(* IEC 61131-3 sources: ml2plc/benchmarks/st (part 26) *)

VAR
    (* Merged variables from all regions *)
    buffer_0 : ARRAY[0..63] OF REAL;
    buffer_1 : ARRAY[0..63] OF REAL;
    buffer_2 : ARRAY[0..63] OF REAL;

    (* Temporary computation variables *)
    i : DINT;
    j : DINT;
    t : DINT;
    sum : REAL;
    (* Computation helpers *)
    max_val : REAL;
    exp_val : REAL;
    exp_sum : REAL;
    (* Spatial loop variables *)
    oc : DINT;
    oh : DINT;
    ow : DINT;
    ic : DINT;
    kh : DINT;
    kw : DINT;
    ih : DINT;
    iw : DINT;
END_VAR

(* Forward pass execution *)

(* Region: r0 [ACYCLIC] *)
(* Acyclic Region r0 *)
(* Layer 0: Fused Linear + RELU *)
FOR j := 0 TO 63 DO
    sum := 0.0;
    FOR i := 0 TO 0 DO
        sum := sum + input_data * weights_0[i * 64 + j];
    END_FOR;
buffer_0[j] := MAX(sum + bias_0[j], 0.0);
END_FOR;

(* Layer 1: Fused Linear + RELU *)
FOR j := 0 TO 63 DO
    sum := 0.0;
    FOR i := 0 TO 63 DO
        sum := sum + buffer_0[i] * weights_1[i * 64 + j];
    END_FOR;
buffer_2[j] := MAX(sum + bias_1[j], 0.0);
END_FOR;

(* Layer 2: MatMul *)
FOR j := 0 TO 63 DO
    sum := 0.0;
    FOR i := 0 TO 63 DO
        sum := sum + buffer_2[i] * weights_2[i * 64 + j];
    END_FOR;
buffer_1[j] := sum;
END_FOR;

(* Layer 3: Add (Bias) *)
FOR i := 0 TO 63 DO
    buffer_2[i] := buffer_1[i] + bias_3[i];
END_FOR;

(* Layer 4: Add (Element-wise) *)
FOR i := 0 TO 63 DO
    buffer_1[i] := buffer_2[i] + buffer_0[i];
END_FOR;

(* Layer 5: Activation (RELU) *)
FOR i := 0 TO 63 DO
    buffer_0[i] := MAX(buffer_1[i], 0.0);
END_FOR;

(* Layer 6: Fused Linear + RELU *)
FOR j := 0 TO 63 DO
    sum := 0.0;
    FOR i := 0 TO 63 DO
        sum := sum + buffer_0[i] * weights_6[i * 64 + j];
    END_FOR;
buffer_2[j] := MAX(sum + bias_6[j], 0.0);
END_FOR;

(* Layer 7: MatMul *)
FOR j := 0 TO 63 DO
    sum := 0.0;
    FOR i := 0 TO 63 DO
        sum := sum + buffer_2[i] * weights_7[i * 64 + j];
    END_FOR;
buffer_1[j] := sum;
END_FOR;

(* Layer 8: Add (Bias) *)
FOR i := 0 TO 63 DO
    buffer_2[i] := buffer_1[i] + bias_8[i];
END_FOR;

(* Layer 9: Add (Element-wise) *)
FOR i := 0 TO 63 DO
    buffer_1[i] := buffer_2[i] + buffer_0[i];
END_FOR;

(* Layer 10: Activation (RELU) *)
FOR i := 0 TO 63 DO
    buffer_0[i] := MAX(buffer_1[i], 0.0);
END_FOR;

(* Layer 11: Fused Linear + RELU *)
FOR j := 0 TO 63 DO
    sum := 0.0;
    FOR i := 0 TO 63 DO
        sum := sum + buffer_0[i] * weights_11[i * 64 + j];
    END_FOR;
buffer_2[j] := MAX(sum + bias_11[j], 0.0);
END_FOR;

(* Layer 12: MatMul *)
FOR j := 0 TO 63 DO
    sum := 0.0;
    FOR i := 0 TO 63 DO
        sum := sum + buffer_2[i] * weights_12[i * 64 + j];
    END_FOR;
buffer_1[j] := sum;
END_FOR;

(* Layer 13: Add (Bias) *)
FOR i := 0 TO 63 DO
    buffer_2[i] := buffer_1[i] + bias_13[i];
END_FOR;

(* Layer 14: Add (Element-wise) *)
FOR i := 0 TO 63 DO
    buffer_1[i] := buffer_2[i] + buffer_0[i];
END_FOR;

(* Layer 15: Activation (RELU) *)
FOR i := 0 TO 63 DO
    buffer_0[i] := MAX(buffer_1[i], 0.0);
END_FOR;

(* Layer 16: Fused Linear + SOFTMAX *)
FOR j := 0 TO 2 DO
    sum := 0.0;
    FOR i := 0 TO 63 DO
        sum := sum + buffer_0[i] * weights_16[i * 3 + j];
    END_FOR;
output_data[j] := sum + bias_16[j];
END_FOR;

(* Softmax: find max *)
max_val := output_data[0];
FOR i := 1 TO 2 DO
    IF output_data[i] > max_val THEN
        max_val := output_data[i];
    END_IF;
END_FOR;

(* Softmax: compute exponentials and sum *)
exp_sum := 0.0;
FOR i := 0 TO 2 DO
    output_data[i] := EXP(output_data[i] - max_val);
    exp_sum := exp_sum + output_data[i];
END_FOR;

(* Softmax: normalize *)
FOR i := 0 TO 2 DO
    output_data[i] := output_data[i] / exp_sum;
END_FOR;

END_FUNCTION_BLOCK
